///////////
// Structure For Battery Racks. Main Operating Data to be saved ( ex: OPC ) .  
//////////
TYPE RackString_SAFT :
STRUCT
	
		MesData		: RackString ;
		Module		: ARRAY[1..CstNbModule_Rack_G] OF  Module ; 
		
     	
	
		

		
		
		
		
		
		
		
	
END_STRUCT
END_TYPE

(* stored: Version 1.1.0.1, ProductVersion 3.1.4024.11
   DUT RackString_SAFT: Id {57ddaec1-5a1b-4e0f-be42-60d49c981777} *)
